# EPICS substitutions: utcaApp/Db/acq.substitutions
file db/scan_task.template {
    {}
}

file db/acq.template {
    {}
}
